// Mitsubishi GX Works2 project: intel   PLC: Q03UDV

PROGRAM MAIN
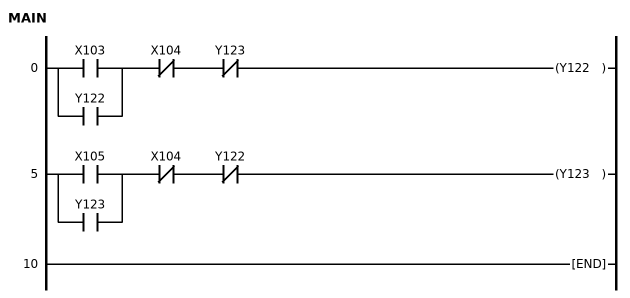
0     LD      X103
      OR      Y122
      ANI     X104
      ANI     Y123
      OUT     Y122
5     LD      X105
      OR      Y123
      ANI     X104
      ANI     Y122
      OUT     Y123
10    END
END_PROGRAM
